FUNCTION_BLOCK SkillFB (* Composite FB wrapping other FBs *)
  (* Standard: 61499-2 *)
  (* Version 1.0, 2021-03-18, AK120569 *)
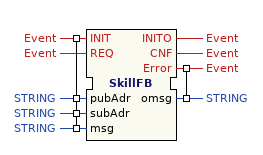
  EVENT_INPUT
    INIT WITH subAdr, pubAdr, msg; (* Initialization Request *)
    REQ; (* Normal Execution Request *)
  END_EVENT
  EVENT_OUTPUT
    INITO; (* Initialization Confirm *)
    CNF; (* Execution Confirmation *)
    Error WITH omsg;
  END_EVENT
  VAR_INPUT
    pubAdr : STRING;
    subAdr : STRING;
    msg : STRING;
  END_VAR
  VAR_OUTPUT
    omsg : STRING;
  END_VAR
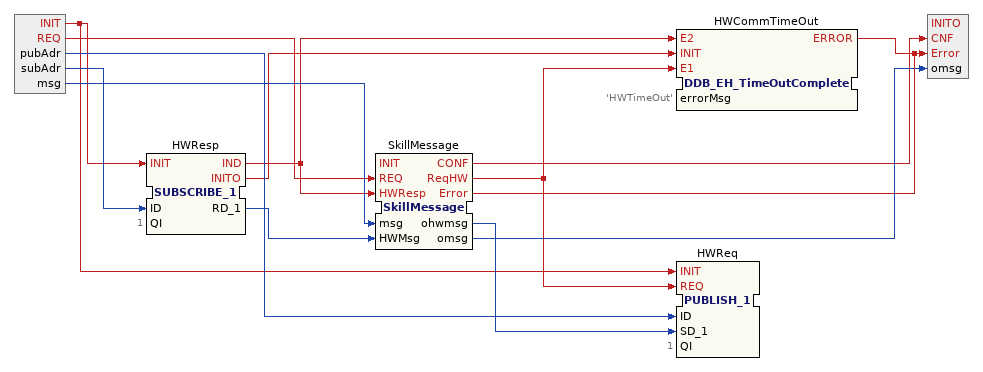
  FBS
    HWReq : PUBLISH_1(QI := 1);
    HWResp : SUBSCRIBE_1(QI := 1);
    HWCommTimeOut : DDB_EH_TimeOutComplete(errorMsg := 'HWTimeOut');
    SkillMessage : SkillMessage;
  END_FBS
  EVENT_CONNECTIONS
    INIT TO HWReq.INIT;
    INIT TO HWResp.INIT;
    HWCommTimeOut.ERROR TO Error;
    HWResp.IND TO HWCommTimeOut.E2;
    HWResp.INITO TO HWCommTimeOut.INIT;
    REQ TO SkillMessage.REQ;
    HWResp.IND TO SkillMessage.HWResp;
    SkillMessage.Error TO Error;
    SkillMessage.ReqHW TO HWCommTimeOut.E1;
    SkillMessage.ReqHW TO HWReq.REQ;
    SkillMessage.CONF TO CNF;
  END_CONNECTIONS
  DATA_CONNECTIONS
    pubAdr TO HWReq.ID;
    subAdr TO HWResp.ID;
    HWResp.RD_1 TO SkillMessage.HWMsg;
    msg TO SkillMessage.msg;
    SkillMessage.ohwmsg TO HWReq.SD_1;
    SkillMessage.omsg TO omsg;
  END_CONNECTIONS
END_FUNCTION_BLOCK
